(* LS Electric XG5000 project: Trafic_Light_Control *)
(* PLC LSPLC *)

PROGRAM NewProgram (* task: Scan Program *)
VAR
    GreenLight AT %QX0.0.10 : BOOL;
    Green_1 AT %QX0.0.6 : BOOL;
    INST : TON;
    ON AT %IX0.0.0 : BOOL;
    RedLight AT %QX0.0.8 : BOOL;
    Red_1 AT %QX0.0.5 : BOOL;
    S1 : BOOL;
    S2 : BOOL;
    S3 : BOOL;
    TIemer_34 : TON;
    Timer1 : TON;
    Timer_2 : TON;
    Timer_3 : TON;
    Timer_34 : TMR;
    Timer_35 : TON;
    YellowLight AT %QX0.0.9 : BOOL;
    Yellow_1 AT %QX0.0.7 : BOOL;
END_VAR

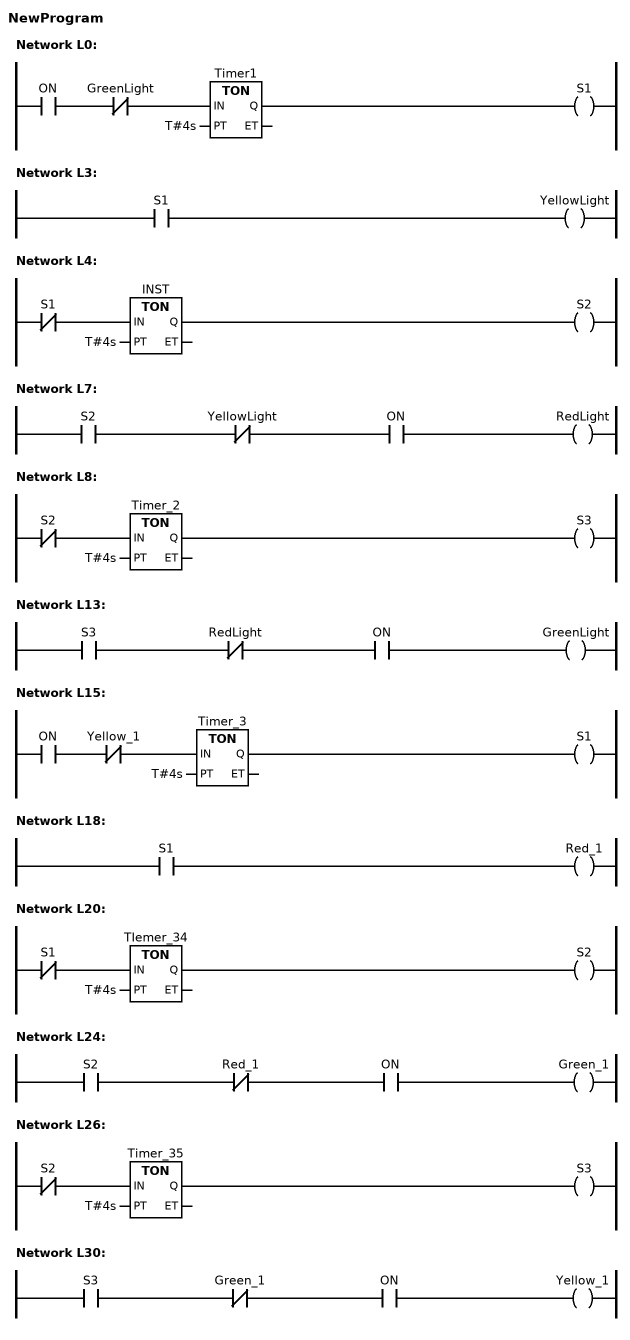
(* Rung L0 *)
Timer1(IN := ON AND NOT GreenLight, PT := T#4s);
S1 := Timer1.Q;
(* Rung L3 *)
YellowLight := S1;
(* Rung L4 *)
INST(IN := NOT S1, PT := T#4s);
S2 := INST.Q;
(* Rung L7 *)
RedLight := S2 AND NOT YellowLight AND ON;
(* Rung L8 *)
Timer_2(IN := NOT S2, PT := T#4s);
S3 := Timer_2.Q;
(* Rung L13 *)
GreenLight := S3 AND NOT RedLight AND ON;
(* Rung L15 *)
Timer_3(IN := ON AND NOT Yellow_1, PT := T#4s);
S1 := Timer_3.Q;
(* Rung L18 *)
Red_1 := S1;
(* Rung L20 *)
TIemer_34(IN := NOT S1, PT := T#4s);
S2 := TIemer_34.Q;
(* Rung L24 *)
Green_1 := S2 AND NOT Red_1 AND ON;
(* Rung L26 *)
Timer_35(IN := NOT S2, PT := T#4s);
S3 := Timer_35.Q;
(* Rung L30 *)
Yellow_1 := S3 AND NOT Green_1 AND ON;
END_PROGRAM